(* A dynamic array that holds data of multiple types and can grow or shrink at run time. *)
{attribute 'enable_dynamic_creation'}
{attribute 'no_assign'}
FUNCTION_BLOCK FB_Array_List EXTENDS FB_Collection IMPLEMENTS I_List, I_Generic_List
VAR
	pData 		: POINTER TO ST_GENERIC;
END_VAR
VAR CONSTANT
	//{warning disable C0228}
	stData 		: ST_GENERIC := (TypeClass := __SYSTEM.TYPE_CLASS.TYPE_NONE);
END_VAR

(* Checks of list is empty.*)
PROPERTY _Is_Empty : BOOL
GET
_Is_Empty := THIS^.nCount = 0;
END_GET
END_PROPERTY

// Adds an item to the end of the list
METHOD Add_Back : I_List
VAR_INPUT
	Item 	: ANY; // Item to store in list
END_VAR
VAR_OUTPUT
	bSuccess : BOOL;
END_VAR
Add_Back := THIS^;
IF THIS^._Is_Empty THEN THIS^.FB_init(FALSE,FALSE, 1); THIS^.Set(Item, 0, bSuccess => bSuccess); RETURN; END_IF
THIS^.Resize(THIS^._Count+1);
THIS^.Free_Value(THIS^.pData[THIS^._Count-1]);
THIS^.pData[THIS^._Count-1] := THIS^.Malloc_Value(Item);
THIS^.CopyValueTo(THIS^.pData[THIS^._Count-1], Item);
bSuccess := TRUE;
END_METHOD

// Adds an item at the front of the list
METHOD Add_Front : I_List
VAR_INPUT
	Item 	 : ANY; // Item to store in list
END_VAR
VAR_OUTPUT
	bSuccess : BOOL;
END_VAR
VAR
	pOld_Data : POINTER TO ST_GENERIC;
	i : DINT;
END_VAR
Add_Front := THIS^;
IF THIS^._Is_Empty THEN THIS^.FB_init(FALSE,FALSE, 1); THIS^.Set(Item, 0, bSuccess => bSuccess); RETURN; END_IF

pOld_Data := THIS^.pData;
THIS^.pData := THIS^.Malloc_Array(THIS^._Count+1);

FOR i := 1 TO THIS^._Count DO
	THIS^.pData[i] := THIS^.Malloc_Value(pOld_Data[i-1]);
	THIS^.CopyValueTo(THIS^.pData[i], pOld_Data[i-1]);
	THIS^.Free_Value(pOld_Data[i-1]);
	END_FOR
__DELETE(pOld_Data);
THIS^.Set(Item, 0);
THIS^.IncrementCount();
bSuccess := TRUE;
END_METHOD

// Empties/Clears/Deletes every item in the list
METHOD Clear
VAR
	i : DINT;
END_VAR
IF NOT(THIS^._Is_Empty) THEN 
	FOR i := 0 TO THIS^._Count - 1 DO THIS^.Free_Value(THIS^.pData[i]); END_FOR
	__DELETE(THIS^.pData); 
	THIS^.nCount := 0; 
	END_IF
END_METHOD

(* Checks if item is contained in list *)
METHOD Contains : BOOL
VAR_INPUT
	Item : ANY; // Item to find in list
END_VAR
THIS^.Find(Item, bSuccess => Contains);
END_METHOD

// Copy data from source memory space to desination memory space
METHOD PROTECTED CopyValueTo
VAR_INPUT
	Dest, Src 	: T_Generic;
END_VAR
MEMMOVE(Dest.pValue, Src.pValue, TO_UDINT(Src.diSize));
END_METHOD

// Decrement list size by 1.
METHOD PROTECTED DecrementCount
THIS^.nCount := THIS^.nCount - 1;
END_METHOD

// Raises an expection if list is empty
METHOD PROTECTED EmptyListException : BOOL
VAR_INPUT
END_VAR
IF THIS^._Is_Empty THEN
	stError.bSTATUS := TRUE;
	stError.nCODE 	:= 2936;
	stError.sSOURCE := 'List is empty';
ELSE
	This^.ClearException();
	END_IF
EmptyListException := stError.bSTATUS;
END_METHOD

METHOD FB_exit : BOOL
VAR_INPUT
	bInCopyCode : BOOL; // if TRUE, the exit method is called for exiting an instance that is copied afterwards (online change).
END_VAR
THIS^.Clear();
END_METHOD

METHOD FB_init : BOOL
VAR_INPUT
	bInitRetains 	: BOOL; 		// if TRUE, the retain variables are initialized (warm start / cold start)
	bInCopyCode 	: BOOL; 		// if TRUE, the instance afterwards gets moved into the copy code (online change)
	nLength 		: T_Capacity;	// Length to initialise array with.
END_VAR
VAR
	i, nByte_Size 	: DINT;
END_VAR
THIS^.Clear();
IF nLength <= 0 THEN RETURN; END_IF
THIS^.nCount := nLength;
THIS^.pData := THIS^.Malloc_Array(nLength);
END_METHOD

// Find the location of an item in list.
METHOD Find : I_List
VAR_INPUT
	Item 		: ANY; // Item to find in list
END_VAR
VAR_OUTPUT
	nIndex		: T_Capacity; //Location of item in list 
	bSuccess 	: BOOL;
END_VAR
VAR
	i : DINT;
	n : DINT := -1;
END_VAR
Find := THIS^;
IF THIS^.EmptyListException() THEN nIndex := -1; RETURN; END_IF
FOR i := 0 TO THIS^._Count-1 DO
	IF (THIS^.pData[i].pValue = 0) 					 THEN CONTINUE; END_IF
	IF (Item.TypeClass <> THIS^.pData[i].TypeClass) THEN CONTINUE; END_IF
	IF (Item.pValue^ <> THIS^.pData[i].pValue^) 	 THEN CONTINUE; END_IF
	
	CASE Item.TypeClass OF
		__SYSTEM.TYPE_CLASS.TYPE_STRING:
			IF LEN2(Item.pValue) <> LEN2(THIS^.pData[i].pValue) THEN CONTINUE; END_IF
			n := MEMCMP(Item.pValue, THIS^.pData[i].pValue, LEN2(THIS^.pData[i].pValue)+1);
				
		__SYSTEM.TYPE_CLASS.TYPE_WSTRING:
			IF WLEN2(Item.pValue) <> WLEN2(THIS^.pData[i].pValue) THEN CONTINUE; END_IF
			n := MEMCMP(Item.pValue, THIS^.pData[i].pValue, (WLEN2(THIS^.pData[i].pValue)*SIZEOF(WORD))+1);
	ELSE
		IF (Item.diSize <> THIS^.pData[i].diSize) THEN CONTINUE; END_IF	
		n := MEMCMP(Item.pValue, THIS^.pData[i].pValue, TO_UDINT(Item.diSize));
		END_CASE
		IF n = 0 THEN nIndex := i; bSuccess := TRUE; RETURN; END_IF
	END_FOR
nIndex := -1;
END_METHOD

// Deletes/frees Generic value's value from memory
METHOD PROTECTED Free_Value
VAR_INPUT
	Variable : T_Generic;
END_VAR
IF Variable.pValue = 0 THEN RETURN; END_IF
__DELETE(Variable.pValue);
END_METHOD

// Gets item at specified location;
METHOD Get : I_List
VAR_INPUT
	Return_Item 	: ANY;  // Variable to store requested node value
	nIndex 			: T_Capacity; // Location of node
END_VAR
VAR_OUTPUT
	bSuccess 		: BOOL;
END_VAR
Get := THIS^;
IF THIS^.EmptyListException() OR THIS^.OutOfBoundsException(nIndex) THEN RETURN; END_IF
IF THIS^.TypeMismatchException(Return_Item, THIS^.pData[nIndex]) THEN RETURN; END_IF
THIS^.CopyValueTo(Return_Item, THIS^.pData[nIndex]);
bSuccess := TRUE;
END_METHOD

// Gets item at the front of the list 
METHOD Get_First : I_List
VAR_INPUT
	Return_Item 	: ANY; // Variable to store returned item
END_VAR
VAR_OUTPUT
	bSuccess : BOOL;
END_VAR
Get_First := THIS^;
THIS^.Get(Return_Item, 0, bSuccess => bSuccess);
END_METHOD

// Gets a value from a list in it's generic form.
// (* Use carefully as this contains the pointer of the actual value in the collection. *)
// If you wish to use this it is recommeded you create a copy of the returned value using MEMMOVE or MEMCPY
METHOD Get_Generic : I_Generic_List
VAR_INPUT
	nIndex 		: T_Capacity; 	// Location of item
END_VAR
VAR_OUTPUT
	Return_Item : T_Generic;  	// Variable to store returned item
	bSuccess 	: BOOL;
END_VAR
Get_Generic := THIS^;
IF THIS^.EmptyListException() OR THIS^.OutOfBoundsException(nIndex) THEN RETURN; END_IF
Return_Item := THIS^.pData[nIndex];
bSuccess := TRUE;
END_METHOD

// Gets item at the back of the list 
METHOD Get_Last : I_List
VAR_INPUT
	Return_Item 	: ANY; // Variable to store returned item
END_VAR
VAR_OUTPUT
	bSuccess : BOOL;
END_VAR
Get_Last := THIS^;
THIS^.Get(Return_Item, THIS^._Count - 1, bSuccess => bSuccess);
END_METHOD

// Returns item as a string, if type to string conversion is supported
METHOD Get_Value_As_String : I_List
VAR_INPUT
	nIndex	: T_Capacity; // Location of item
END_VAR
VAR_OUTPUT
	sItem 	: T_MaxString; // Variable to store returned item
END_VAR
Get_Value_As_String := THIS^;
IF THIS^.EmptyListException() OR THIS^.OutOfBoundsException(nIndex) THEN sItem := 'ERR: List is Empty or index Out of Bounds'; RETURN; END_IF
sItem := THIS^.pData[nIndex].sValue;
END_METHOD

METHOD PROTECTED GetValueAsString : T_MaxString
VAR_INPUT
	 Value : T_Generic;
END_VAR
VAR	
	pBool			: POINTER TO BOOL;
    pByte			: POINTER TO BYTE;
    pWord			: POINTER TO WORD;
    pDWord			: POINTER TO DWORD;
    pLWord			: POINTER TO LWORD;
    pSint			: POINTER TO SINT;
    pInt			: POINTER TO INT;
    pDint			: POINTER TO DINT;
    pLint			: POINTER TO LINT;
    pUSint			: POINTER TO USINT;
    pUInt			: POINTER TO UINT;
    pUDint			: POINTER TO UDINT;
    pULint			: POINTER TO ULINT;
    pReal			: POINTER TO REAL;
    pLReal			: POINTER TO LREAL;
    pString			: POINTER TO STRING(255);
    pWString		: POINTER TO WSTRING;
    pTime			: POINTER TO TIME;
    pDate			: POINTER TO DATE;
    pDate_And_Time	: POINTER TO DATE_AND_TIME;
    pTime_Of_Day	: POINTER TO TIME_OF_DAY;
    pPointer		: PVOID;
	pLTime 			: POINTER TO LTIME;
END_VAR
IF Value.pValue = 0 THEN GetValueAsString := 'NULL'; RETURN; END_IF;

CASE Value.TypeClass OF 
	__SYSTEM.TYPE_CLASS.TYPE_BOOL:
		pBool := Value.pValue;
		GetValueAsString := TO_STRING(pBool^);
		
    __SYSTEM.TYPE_CLASS.TYPE_BYTE:
		pByte := Value.pValue;
		GetValueAsString := TO_STRING(pByte^);
		
    __SYSTEM.TYPE_CLASS.TYPE_WORD:
		pWord := Value.pValue;
		GetValueAsString := TO_STRING(pWord^);
		
    __SYSTEM.TYPE_CLASS.TYPE_DWORD:
		pDWord := Value.pValue;
		GetValueAsString := TO_STRING(pDWord^);
		
    __SYSTEM.TYPE_CLASS.TYPE_LWORD:
		pLWord := Value.pValue;
		GetValueAsString := TO_STRING(pLWord^);
		
    __SYSTEM.TYPE_CLASS.TYPE_SINT:
		pSint := Value.pValue;
		GetValueAsString := TO_STRING(pSint^);
		
    __SYSTEM.TYPE_CLASS.TYPE_INT:
		pInt := Value.pValue;
		GetValueAsString := TO_STRING(pInt^);
		
    __SYSTEM.TYPE_CLASS.TYPE_DINT:
		pDint := Value.pValue;
		GetValueAsString := TO_STRING(pDint^);
		
    __SYSTEM.TYPE_CLASS.TYPE_LINT:
		pLint := Value.pValue;
		GetValueAsString := TO_STRING(pLint^);
		
    __SYSTEM.TYPE_CLASS.TYPE_USINT:
		pUSint := Value.pValue;
		GetValueAsString := TO_STRING(pUSint^);
		
    __SYSTEM.TYPE_CLASS.TYPE_UINT:
		pUInt := Value.pValue;
		GetValueAsString := TO_STRING(pUInt^);
		
    __SYSTEM.TYPE_CLASS.TYPE_UDINT:
		pUDint := Value.pValue;
		GetValueAsString := TO_STRING(pUDint^);
		
    __SYSTEM.TYPE_CLASS.TYPE_ULINT:
		pULint := Value.pValue;
		GetValueAsString := TO_STRING(pULint^);
		
   __SYSTEM.TYPE_CLASS.TYPE_REAL:
		pReal := Value.pValue;
		GetValueAsString := TO_STRING(pReal^);
		
    __SYSTEM.TYPE_CLASS.TYPE_LREAL:
		pLReal := Value.pValue;
		GetValueAsString := TO_STRING(pLReal^);
		
    __SYSTEM.TYPE_CLASS.TYPE_STRING:
		pString := Value.pValue;
		GetValueAsString := TO_STRING(pString^);
		
   __SYSTEM.TYPE_CLASS.TYPE_WSTRING:
		pWString := Value.pValue;
		GetValueAsString := TO_STRING(pWString^);
		
    __SYSTEM.TYPE_CLASS.TYPE_TIME:
		pTime := Value.pValue;
		GetValueAsString := TO_STRING(pTime^);
		
    __SYSTEM.TYPE_CLASS.TYPE_DATE:
		pDate := Value.pValue;
		GetValueAsString := TO_STRING(pDate^);
		
    __SYSTEM.TYPE_CLASS.TYPE_DATEANDTIME:
		pDate_And_Time := Value.pValue;
		GetValueAsString := TO_STRING(pDate_And_Time^);
		
    __SYSTEM.TYPE_CLASS.TYPE_TIMEOFDAY:
		pTime_Of_Day := Value.pValue;
		GetValueAsString := TO_STRING(pTime_Of_Day^);
	
	__SYSTEM.TYPE_CLASS.TYPE_POINTER:
		GetValueAsString := TO_STRING(Value.pValue);
		
	__SYSTEM.TYPE_CLASS.TYPE_LTIME:
		pLTime := Value.pValue;
		GetValueAsString := TO_STRING(pLTime^);
ELSE
	GetValueAsString := 'TYPE TO STRING CONVERSION NOT SUPPORTED BY THIS TYPE'; 
END_CASE
END_METHOD

// Increments list size by 1
METHOD PROTECTED IncrementCount
VAR_INPUT
END_VAR
THIS^.nCount := THIS^.nCount + 1;
END_METHOD

// Adds new item to list at specified location, if index = 0, item will be added at the front, if index = count, item will be added at the back
METHOD Insert : I_List
VAR_INPUT
	Item 	: ANY;  		// Item to store in list
	nIndex 	: T_Capacity; // Location of item
END_VAR
VAR_OUTPUT
	bSuccess : BOOL;
END_VAR
VAR
	pOld_Data 	: POINTER TO T_Generic;
	i 			: T_Capacity;
END_VAR
Insert := THIS^;
IF nIndex = 0 THEN THIS^.Add_Front(Item, bSuccess => bSuccess); RETURN; END_IF
IF nIndex = THIS^._Count THEN THIS^.Add_Back(Item, bSuccess => bSuccess); RETURN; END_IF
IF THIS^.OutOfBoundsException(nIndex) THEN RETURN; END_IF

pOld_Data := THIS^.pData;
THIS^.pData := THIS^.Malloc_Array(THIS^._Count+1);
THIS^.IncrementCount();

FOR i := 0 TO nIndex-1 DO
	THIS^.pData[i] := THIS^.Malloc_Value(pOld_Data[i]);
	THIS^.CopyValueTo(THIS^.pData[i], pOld_Data[i]);
	THIS^.Free_Value(pOld_Data[i]);
	END_FOR
	
THIS^.Set(Item, nIndex, bSuccess => bSuccess);
	
FOR i := nIndex+1 TO THIS^._Count-1 DO
	THIS^.pData[i] := THIS^.Malloc_Value(pOld_Data[i-1]);
	THIS^.CopyValueTo(THIS^.pData[i], pOld_Data[i-1]);
	THIS^.Free_Value(pOld_Data[i-1]);
	END_FOR
__DELETE(pOld_Data);
END_METHOD

// Adds new item to list at specified location using the generic form. 
// If index = 0, item will be added at the front, if index = count, item will be added at the back
METHOD Insert_Generic : I_Generic_List
VAR_INPUT
	Item 	: T_Generic;  	// Item to store in list
	nIndex 	: T_Capacity; 			// Location of item
END_VAR
VAR_OUTPUT
	bSuccess : BOOL;
END_VAR
VAR
	pOld_Data 	: POINTER TO T_Generic;
	i 			: T_Capacity;
END_VAR
Insert_Generic := THIS^;

// Add to front
IF nIndex = 0 THEN THIS^.Internal_Add_Front(Item, bSuccess => bSuccess); RETURN; END_IF

// Add to back
IF nIndex = THIS^._Count THEN Internal_Add_Back(Item, bSuccess => bSuccess); RETURN; END_IF

IF THIS^.OutOfBoundsException(nIndex) THEN RETURN; END_IF

pOld_Data := THIS^.pData;
THIS^.pData := THIS^.Malloc_Array(THIS^._Count+1);
THIS^.IncrementCount();

FOR i := 0 TO nIndex-1 DO
	THIS^.pData[i] := THIS^.Malloc_Value(pOld_Data[i]);
	THIS^.CopyValueTo(THIS^.pData[i], pOld_Data[i]);
	THIS^.Free_Value(pOld_Data[i]);
	END_FOR

// Set value
Internal_Set(Item, nIndex, bSuccess => bSuccess);
	
FOR i := nIndex+1 TO THIS^._Count-1 DO
	THIS^.pData[i] := THIS^.Malloc_Value(pOld_Data[i-1]);
	THIS^.CopyValueTo(THIS^.pData[i], pOld_Data[i-1]);
	THIS^.Free_Value(pOld_Data[i-1]);
	END_FOR
__DELETE(pOld_Data);
END_METHOD

// Adds an item to the end of the list
METHOD PROTECTED Internal_Add_Back
VAR_INPUT
	Item 		: T_Generic; // Item to store in list
END_VAR
VAR_OUTPUT
	bSuccess 	: BOOL;
END_VAR
IF THIS^._Is_Empty THEN THIS^.FB_init(FALSE,FALSE, 1); THIS^.Internal_Set(Item, 0, bSuccess => bSuccess); RETURN; END_IF
THIS^.Resize(THIS^._Count+1);
THIS^.Free_Value(THIS^.pData[THIS^._Count-1]);
THIS^.pData[THIS^._Count-1] := THIS^.Malloc_Value(Item);
THIS^.CopyValueTo(THIS^.pData[THIS^._Count-1], Item);
bSuccess := TRUE;
END_METHOD

// Adds an item at the front of the list
METHOD PROTECTED Internal_Add_Front
VAR_INPUT
	Item 	 : ANY; // Item to store in list
END_VAR
VAR_OUTPUT
	bSuccess : BOOL;
END_VAR
VAR
	pOld_Data : POINTER TO ST_GENERIC;
	i : DINT;
END_VAR
IF THIS^._Is_Empty THEN THIS^.FB_init(FALSE,FALSE, 1); THIS^.Internal_Set(Item, 0, bSuccess => bSuccess); RETURN; END_IF

pOld_Data := THIS^.pData;
THIS^.pData := THIS^.Malloc_Array(THIS^._Count+1);

FOR i := 1 TO THIS^._Count DO
	THIS^.pData[i] := THIS^.Malloc_Value(pOld_Data[i-1]);
	THIS^.CopyValueTo(THIS^.pData[i], pOld_Data[i-1]);
	THIS^.Free_Value(pOld_Data[i-1]);
	END_FOR
__DELETE(pOld_Data);
THIS^.Internal_Set(Item, 0);
THIS^.IncrementCount();
bSuccess := TRUE;
END_METHOD

// Adds new item to list in the specified location without resizing list
METHOD PROTECTED Internal_Set
VAR_INPUT
	Item 	: T_Generic; 	// Item to store in list
	nIndex 	: T_Capacity; // Location of item
END_VAR
VAR_OUTPUT
	bSuccess : BOOL;
END_VAR
IF THIS^.OutOfBoundsException(nIndex) OR THIS^.EmptyListException() THEN RETURN; END_IF
THIS^.Free_Value(THIS^.pData[nIndex]);
THIS^.pData[nIndex] := THIS^.Malloc_Value(Item);
THIS^.CopyValueTo(THIS^.pData[nIndex], Item);
bSuccess := TRUE;
END_METHOD

METHOD PROTECTED LessThanZeroException : BOOL
VAR_INPUT
	nIndex : DINT;
END_VAR
IF (nIndex < 0) THEN
	stError.bSTATUS := TRUE;
	stError.nCODE 	:= 5365;
	stError.sSOURCE := 'Out of bounds. Index is less than zero.';
ELSE
	This^.ClearException();
	END_IF
LessThanZeroException := stError.bSTATUS;
END_METHOD

// Allocate memory space for Array of Generics on the heap, returns Pointer to start of Generic Array;
// WARNING!!! Always have a place to store the return otherwise a memory leak will occur.
METHOD PROTECTED Malloc_Array : POINTER TO ST_GENERIC
VAR_INPUT
	nSize : T_Capacity; // Array Size
END_VAR
VAR
	i, nByte_Size: T_Capacity;
END_VAR
VAR CONSTANT
	stData 		: T_Generic_Ex := ();
END_VAR
nByte_Size := SIZEOF(T_Generic_Ex)*nSize;
Malloc_Array := __NEW(BYTE, TO_UDINT(nByte_Size));
END_METHOD

// Allocate memory space for the Generic value's data on the heap, returns Generic;
// WARNING!!! Always have a place to store the return otherwise a memory leak will occur.
METHOD PROTECTED Malloc_Value : ST_GENERIC
VAR_INPUT
	Variable : T_Generic;
END_VAR
Malloc_Value.sValue 	:= THIS^.GetValueAsString(Variable);
Malloc_Value.pValue 	:= __NEW(BYTE, TO_UDINT(Variable.diSize)); // Allocate space in memory to store data value.
Malloc_Value.diSize 	:= Variable.diSize;
Malloc_Value.TypeClass 	:= Variable.TypeClass;
END_METHOD

// Compares memory sizes of 2 addresses. Returns TRUE  and raises error flag if theyre not same size.
METHOD PROTECTED MemCmpErrExpection : BOOL
VAR_INPUT
	pDestAddr,
	pSrcAddr 	: PVOID;
	nSize 		: UDINT;
END_VAR
VAR_INST
	nMemErr : DINT;
END_VAR
nMemErr := MEMCMP(pDestAddr, pSrcAddr, nSize);
IF nMemErr = -1 THEN 
	stError.bSTATUS := TRUE;
	stError.nCODE 	:= 4129;
	stError.sSOURCE := 'Incorrect parameter values. Destination address smaller than source address';
	
ELSIF nMemErr = 0 THEN THIS^.ClearException();
	
ELSIF nMemErr = 1 THEN
	stError.bSTATUS := TRUE;
	stError.nCODE 	:= 4823;
	stError.sSOURCE := 'Incorrect parameter values. Destination address greater that source address';

ELSE
	stError.bSTATUS := TRUE;
	stError.nCODE 	:= 4564;
	stError.sSOURCE := 'Incorrect parameter values. Pointer to destination/source address is NULL or allocated address memory is NULL.';
	END_IF

MemCmpErrExpection := stError.bSTATUS;
END_METHOD

METHOD PROTECTED OutOfBoundsException : BOOL
VAR_INPUT
	nIndex : DINT;
END_VAR
IF (nIndex < 0) OR (nIndex >= THIS^._Count) THEN
	stError.bSTATUS := TRUE;
	stError.nCODE 	:= 5374;
	stError.sSOURCE := 'Out of bounds. You tried to access data outside the range of this list.';
ELSE
	This^.ClearException();
	END_IF
OutOfBoundsException := stError.bSTATUS;
END_METHOD

// Removes item at the front of the list and returns nothing
METHOD Remove : I_List
VAR_OUTPUT
	bSuccess : BOOL;
END_VAR
VAR
	i : DINT;
	pOld_Data 	: POINTER TO ST_GENERIC;
END_VAR
//// New ///
Remove := THIS^;
IF THIS^.EmptyListException() THEN RETURN; END_IF
IF THIS^._Count = 1 THEN THIS^.Clear(); bSuccess := TRUE; RETURN; END_IF;

THIS^.Free_Value(THIS^.pData[0]);
pOld_Data := pData;
pData := THIS^.Malloc_Array(THIS^._Count - 1);
FOR i := 1 TO THIS^._Count - 1 DO
	pData[i-1] := pOld_Data[i];
	END_FOR

__DELETE(pOld_Data);
THIS^.DecrementCount();
bSuccess := TRUE;
END_METHOD

// Remove item at specified location and return nothing
METHOD Remove_At : I_List
VAR_INPUT
	nIndex : T_Capacity; // Location of item
END_VAR
VAR_OUTPUT
	bSuccess : BOOL;
END_VAR
VAR
	i : DINT;
END_VAR
Remove_At := THIS^;
IF THIS^.EmptyListException() THEN RETURN; END_IF
IF THIS^.OutOfBoundsException(nIndex) THEN RETURN; END_IF
IF nIndex = 0 THEN THIS^.Remove(bSuccess => bSuccess); RETURN; END_IF
IF nIndex = THIS^._Count - 1 THEN THIS^.Resize(THIS^._Count - 1, bSuccess => bSuccess); RETURN; END_IF
THIS^.Free_Value(THIS^.pData[nIndex]);
FOR i := nIndex TO THIS^._Count-1 DO THIS^.pData[i] := THIS^.pData[i+1]; END_FOR
THIS^.Resize(THIS^._Count-1, bSuccess => bSuccess);
END_METHOD

// Removes item at the back of the list and returns nothing
METHOD Remove_Last : I_List
VAR_OUTPUT
	bSuccess : BOOL;
END_VAR
Remove_Last := THIS^;
THIS^.Remove_At(THIS^._Count-1, bSuccess => bSuccess);
END_METHOD

// Manually resize list. If list becomes smaller, items on higher locations will be deleted.
METHOD Resize : I_List
VAR_INPUT
	nSize : T_Capacity; // New size of list.
END_VAR
VAR_OUTPUT
	bSuccess : BOOL;
END_VAR
VAR
	pOld_Data 		: POINTER TO ST_GENERIC;
	i,
	nOld_Data_Count, 
	nByte_Size : DINT;
END_VAR
Resize := THIS^;
IF THIS^.LessThanZeroException(nSize) THEN RETURN; END_IF
IF (nSize = 0) THEN THIS^.Clear(); RETURN; END_IF
IF nSize = THIS^._Count THEN RETURN; END_IF

bSuccess := TRUE;

IF THIS^._Is_Empty THEN THIS^.FB_init(FALSE,FALSE, nSize); RETURN; END_IF

pOld_Data 		:= THIS^.pData;
nOld_Data_Count := THIS^._Count;

THIS^.pData := THIS^.Malloc_Array(nSize);

FOR i := 0 TO nSize - 1 DO
	IF (i = nOld_Data_Count) AND (nSize > nOld_Data_Count) THEN EXIT; END_IF
	THIS^.pData[i] := THIS^.Malloc_Value(pOld_Data[i]);
	THIS^.CopyValueTo(THIS^.pData[i], pOld_Data[i]);
	THIS^.Free_Value(pOld_Data[i]);
	END_FOR
__DELETE(pOld_Data);
THIS^.nCount := nSize;

bSuccess := TRUE;
END_METHOD

// Reverses the order of items in the list
METHOD Reverse : I_List
VAR_OUTPUT
	bSuccess : BOOL;
END_VAR
VAR
	pOld_Data 	: POINTER TO ST_GENERIC;
	nByte_Size 	: DINT;
	i			: DINT;
END_VAR
Reverse := THIS^;
IF THIS^.EmptyListException() THEN RETURN; END_IF
IF THIS^._Count = 1 THEN RETURN; END_IF

pOld_Data 	:= THIS^.pData;

THIS^.pData := THIS^.Malloc_Array(THIS^._Count);

FOR i:= 0 TO THIS^._Count - 1 DO
	THIS^.pData[i] := THIS^.Malloc_Value(pOld_Data[(THIS^._Count-1)-i]);
	THIS^.CopyValueTo(THIS^.pData[i], pOld_Data[(THIS^._Count-1)-i]);
	THIS^.Free_Value(pOld_Data[(THIS^._Count-1)-i]);
	END_FOR
__DELETE(pOld_Data);

bSuccess := TRUE;
END_METHOD

// Adds new item to list in the specified location without resizing list
METHOD Set : I_List
VAR_INPUT
	Item 	: ANY; 	// Item to store in list
	nIndex 	: T_Capacity; // Location of item
END_VAR
VAR_OUTPUT
	bSuccess : BOOL;
END_VAR
Set := THIS^;
IF THIS^.OutOfBoundsException(nIndex) OR THIS^.EmptyListException() THEN RETURN; END_IF
THIS^.Free_Value(THIS^.pData[nIndex]);
THIS^.pData[nIndex] := THIS^.Malloc_Value(Item);
THIS^.CopyValueTo(THIS^.pData[nIndex], Item);
bSuccess := TRUE;
END_METHOD

(* Set value of __SYSTEM.Anytype variable *)
METHOD PROTECTED SetValue
VAR_INPUT
	Variable	: T_Generic;
	Value 		: USINT; // Character/byte to set.
END_VAR
MEMSET(Variable.pValue, Value, TO_UDINT(Variable.diSize));
END_METHOD

METHOD TypeMismatchException : BOOL
VAR_INPUT
	Dest,
	Src 	: __SYSTEM.AnyType;
END_VAR
IF Dest.diSize <> Src.diSize THEN
	stError.bSTATUS := TRUE;
	stError.nCODE 	:= 3172;
	stError.sSOURCE := 'Type mismatch. Byte sizes are not the same';
ELSIF Dest.TypeClass <> Src.TypeClass THEN
	stError.bSTATUS := TRUE;
	stError.nCODE 	:= 3172;
	stError.sSOURCE := 'Type mismatch. Type classes are not the same';
ELSE
	THIS^.ClearException();
END_IF
TypeMismatchException := stError.bSTATUS;
END_METHOD

END_FUNCTION_BLOCK

(* stored: Version 1.1.0.1, ProductVersion 3.1.4024.4
   POU FB_Array_List: Id {a252c2ec-d0f6-4cde-8a10-64c6a5e5d19c}, SpecialFunc None
   Folder Exceptions: Id {b026e345-1815-4332-aa85-b3b8117ca159}
   Folder Protected: Id {0ff05d1a-aac3-45fd-92b2-4aecc5c60331}
   Property _Is_Empty: Id {1f35d022-a163-4ed1-81df-d65862dc4a55}
   Get Get: Id {1e27ff54-0d40-488d-bd53-aed4e6cf41e4}
   Method Add_Back: Id {ef4b505f-7aac-4528-b0bf-586d99faa3ff}
   Method Add_Front: Id {0bc84416-1488-4eef-8214-d1f6167807cf}
   Method Clear: Id {782ff445-bf94-4cab-a432-24264a332ea0}
   Method Contains: Id {e09b857a-be50-4588-9fc9-80fa1ed32c65}
   Method CopyValueTo: Id {3eb59317-2002-4c87-860f-e39da026ce34}
   Method DecrementCount: Id {7c4a392c-f27f-4d14-9f0c-613244e78171}
   Method EmptyListException: Id {204a931b-5eac-4f15-a45e-b95440a28a67}
   Method FB_exit: Id {5d9f1864-fee5-4a4c-83b5-9eb706c524ef}
   Method FB_init: Id {ca4a4ec6-058d-46a3-b64e-292b088adb51}
   Method Find: Id {a97433ff-54cd-4691-9512-79e419276055}
   Method Free_Value: Id {05279f32-d0ee-41c0-9cc7-71b95982b7dc}
   Method Get: Id {25fd987c-dee3-4583-86b8-248b2ab2bf61}
   Method Get_First: Id {12998406-1d18-4d2c-877f-c1f8eecd69bd}
   Method Get_Generic: Id {f1887775-34bc-4273-94a3-243ef6085010}
   Method Get_Last: Id {6f54537d-2632-4a8b-8be1-1b8ac39476b1}
   Method Get_Value_As_String: Id {cde62b5e-c798-40ce-bc7c-7963b1e8ded9}
   Method GetValueAsString: Id {f6f987c3-de6b-4f4b-97da-c183d60ec391}
   Method IncrementCount: Id {5ff55ca3-134c-45a2-b380-8afc2eb26ad5}
   Method Insert: Id {98b1b92c-0e96-4d1b-a639-11be5f9adfe9}
   Method Insert_Generic: Id {7b0855f3-dfce-4e11-8911-c0e1111a2cde}
   Method Internal_Add_Back: Id {1c3cbd70-0918-4952-a44a-0cb09816860d}
   Method Internal_Add_Front: Id {5514d0a2-358f-4871-ad7d-9328c28b1bb1}
   Method Internal_Set: Id {7303e032-dbd4-4be1-915f-58ce898b3c75}
   Method LessThanZeroException: Id {046b4e97-9c09-48a2-b949-b080669b924e}
   Method Malloc_Array: Id {3a8df518-1cde-4a08-a734-3e969895273b}
   Method Malloc_Value: Id {a266aa76-ae8a-49dc-9b16-aebbf468ae2f}
   Method MemCmpErrExpection: Id {ac667bb1-a17d-4ac2-9976-a489765a9841}
   Method OutOfBoundsException: Id {5d8b7f07-d3ff-46eb-9596-48b1d35f67fa}
   Method Remove: Id {ef5542aa-ad88-4010-9958-dfc7d8f994e0}
   Method Remove_At: Id {69309f49-923b-4eee-9ed3-911b01ac9825}
   Method Remove_Last: Id {a5284481-503c-4df6-8ca8-53af4dfc0568}
   Method Resize: Id {7f19a3c8-ac71-4ec2-925a-410d4a5ab311}
   Method Reverse: Id {c7bb1663-8a1d-412d-ac93-00cfb818cee8}
   Method Set: Id {d97a48c2-c0c8-43e0-aaa4-302f9b0b411c}
   Method SetValue: Id {b4066bb1-e012-4222-860e-fe69e5d3f8c2}
   Method TypeMismatchException: Id {66bfd727-608e-4d36-aa02-41ebf1a85296} *)
